// TIA Portal V16 export
// export: Created 2023-03-29T11:04:44.0584651Z, ExportSetting WithDefaults, DisplayName Totally Integrated Automation Portal, DisplayVersion V16 Update 6, DisplayName TIA Portal Version Control Interface, DisplayVersion V16 Update 2, DisplayName TIA Portal Openness, DisplayVersion V16 Update 6, DisplayName STEP 7 Professional, DisplayVersion V16 Update 6, DisplayName STEP 7 Safety, DisplayVersion V16, DisplayName WinCC Advanced, DisplayVersion V16 Update 6
FUNCTION_BLOCK "Kontrola przyrostu ciśnieniea"   // FB3, LAD
TITLE = Kalkulacja przyrostu ciśnienia w czasie
{ S7_Optimized_Access := 'TRUE' }
AUTHOR : RTecmer
FAMILY : PID
VERSION : 0.1
// Funkcja ustala czy następuje przyrost ciśnienia, spadek, równowaga. Pomiar dokonywany jest w ustalonym czasie. W zależności od wyliceń ustawiany jest znacznik, który w funkcji Switch_Motor_Extra dopuszcza lub blokuje uruchomienie dodatkowej pompy
// stored: AutoNumber true, IsIECCheckEnabled false, IsRetainMemResEnabled false, MemoryReserve 500, SetENOAutomatically false, UDAEnableTagReadback false
   VAR_INPUT
      "50Hz" : Bool;   // Znacznik 50Hz
      "Set_O2-PID" : Real;   // Zadana wartość ciśnienia [bar]
      Current_bar_1 : Real;   // aktualne ciśnienie
   END_VAR
   VAR_OUTPUT
      Increase_in_value : Bool;   // Wzwrost wartości bar w jednostce czasu
   END_VAR
   VAR_IN_OUT
      Edge1_Hz : Bool;   // Pamięć zbocza dla pierwszego odczytu
      Edge2_Hz : Bool;   // Pamięć zbocza dla drugiego odczytu
      Data_sek_1 : Int;   // Licznik sekund dla pierwszego odczytu
      Data_sek_2 : Int;   // Licznik sekund dla drugiego odczytu
      Pause_1 : Bool;   // Wstrzymanie dla pierwszego czasu
      Pause_2 : Bool;   // wstrzymanie dla drugiego czasu
   END_VAR
   VAR_TEMP   // added for the SCL form of the ladder/FBD networks
      _w1 : Bool;
      _w2 : Bool;
   END_VAR
BEGIN

REGION Network 1: Wstrzymanie dla pierwszego czasu
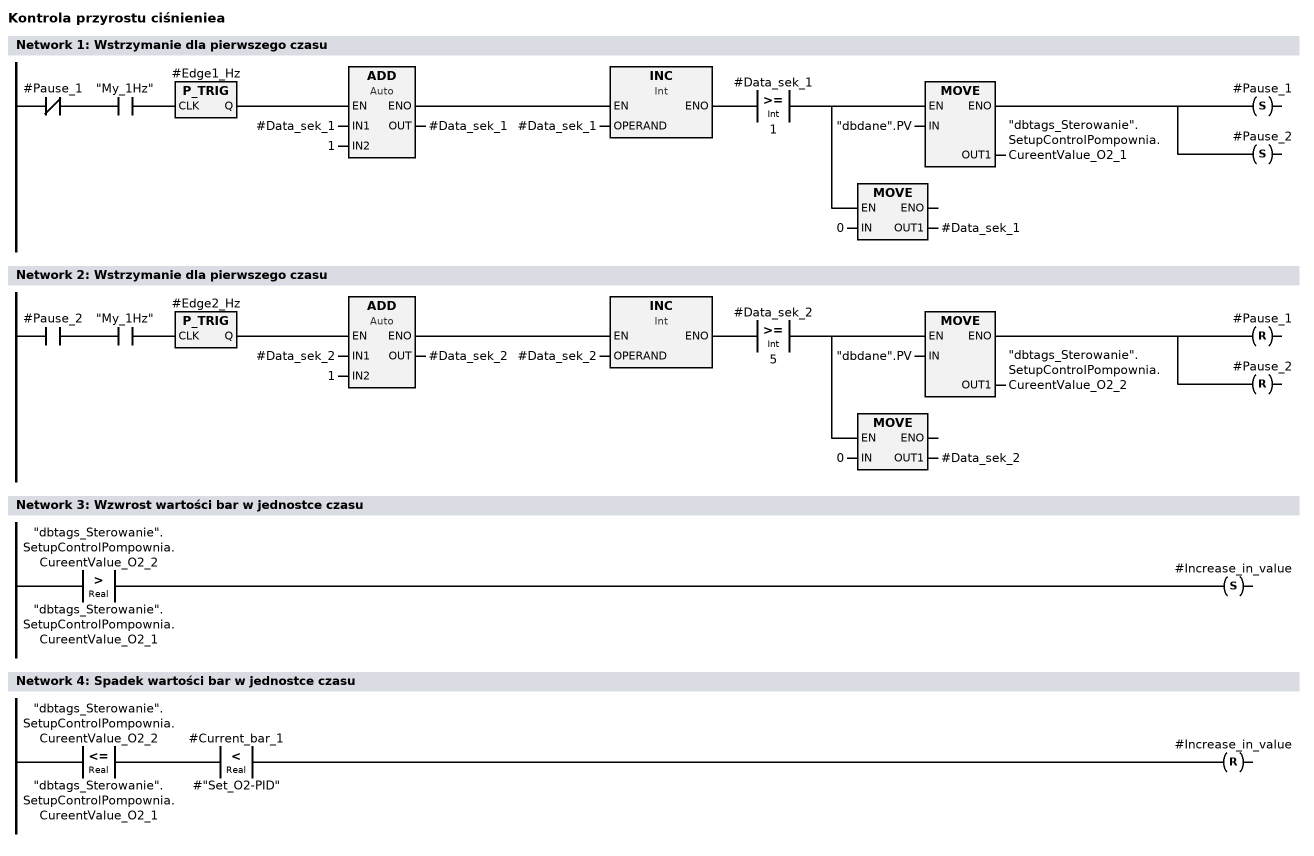
   RUNG wire#powerrail
      I_Contact( #Pause_1 )
      Contact( "My_1Hz" )
      P_Trig( #Edge1_Hz )
      { S7_GenerateENO := "TRUE" } Add(in1 := #Data_sek_1, in2 := 1, out => #Data_sek_1)
      { S7_Templates := "DestType := Int"; S7_GenerateENO := "TRUE" } Inc( #Data_sek_1 )
      { S7_Templates := "SrcType := Int" } GE_Contact(in1 := #Data_sek_1, in2 := 1)
      wire#w1
      { S7_GenerateENO := "TRUE" } Move(in := "dbdane".PV, out1 => "dbtags_Sterowanie".SetupControlPompownia.CureentValue_O2_1)
      wire#w2
      S_Coil( #Pause_1 )
   END_RUNG
   RUNG wire#w2
      S_Coil( #Pause_2 )
   END_RUNG
   RUNG wire#w1
      { S7_GenerateENO := "TRUE" } Move(in := 0, out1 => #Data_sek_1)
   END_RUNG
   // the same network as SCL:
   // ENO of a box is taken as its EN; it also drops when the box reports an error
   #_w1 := NOT #Pause_1 AND "My_1Hz";
   #_w2 := #_w1 AND NOT #Edge1_Hz;   // rising edge
   #Edge1_Hz := #_w1;
   IF #_w2 THEN
       #Data_sek_1 := #Data_sek_1 + 1;
       #Data_sek_1 := #Data_sek_1 + 1;
   END_IF;
   IF #_w2 AND (#Data_sek_1 >= 1) THEN
       "dbtags_Sterowanie".SetupControlPompownia.CureentValue_O2_1 := "dbdane".PV;
       #Pause_1 := TRUE;
       #Pause_2 := TRUE;
       #Data_sek_1 := 0;
   END_IF;
END_REGION

REGION Network 2: Wstrzymanie dla pierwszego czasu
   RUNG wire#powerrail
      Contact( #Pause_2 )
      Contact( "My_1Hz" )
      P_Trig( #Edge2_Hz )
      { S7_GenerateENO := "TRUE" } Add(in1 := #Data_sek_2, in2 := 1, out => #Data_sek_2)
      { S7_Templates := "DestType := Int"; S7_GenerateENO := "TRUE" } Inc( #Data_sek_2 )
      { S7_Templates := "SrcType := Int" } GE_Contact(in1 := #Data_sek_2, in2 := 5)
      wire#w1
      { S7_GenerateENO := "TRUE" } Move(in := "dbdane".PV, out1 => "dbtags_Sterowanie".SetupControlPompownia.CureentValue_O2_2)
      wire#w2
      R_Coil( #Pause_1 )
   END_RUNG
   RUNG wire#w2
      R_Coil( #Pause_2 )
   END_RUNG
   RUNG wire#w1
      { S7_GenerateENO := "TRUE" } Move(in := 0, out1 => #Data_sek_2)
   END_RUNG
   // the same network as SCL:
   // ENO of a box is taken as its EN; it also drops when the box reports an error
   #_w1 := #Pause_2 AND "My_1Hz";
   #_w2 := #_w1 AND NOT #Edge2_Hz;   // rising edge
   #Edge2_Hz := #_w1;
   IF #_w2 THEN
       #Data_sek_2 := #Data_sek_2 + 1;
       #Data_sek_2 := #Data_sek_2 + 1;
   END_IF;
   IF #_w2 AND (#Data_sek_2 >= 5) THEN
       "dbtags_Sterowanie".SetupControlPompownia.CureentValue_O2_2 := "dbdane".PV;
       #Pause_1 := FALSE;
       #Pause_2 := FALSE;
       #Data_sek_2 := 0;
   END_IF;
END_REGION

REGION Network 3: Wzwrost wartości bar w jednostce czasu
   RUNG wire#powerrail
      { S7_Templates := "SrcType := Real" } GT_Contact(in1 := "dbtags_Sterowanie".SetupControlPompownia.CureentValue_O2_2, in2 := "dbtags_Sterowanie".SetupControlPompownia.CureentValue_O2_1)
      S_Coil( #Increase_in_value )
   END_RUNG
   // the same network as SCL:
   IF "dbtags_Sterowanie".SetupControlPompownia.CureentValue_O2_2 > "dbtags_Sterowanie".SetupControlPompownia.CureentValue_O2_1 THEN
       #Increase_in_value := TRUE;
   END_IF;
END_REGION

REGION Network 4: Spadek wartości bar w jednostce czasu
   RUNG wire#powerrail
      { S7_Templates := "SrcType := Real" } LE_Contact(in1 := "dbtags_Sterowanie".SetupControlPompownia.CureentValue_O2_2, in2 := "dbtags_Sterowanie".SetupControlPompownia.CureentValue_O2_1)
      { S7_Templates := "SrcType := Real" } LT_Contact(in1 := #Current_bar_1, in2 := #"Set_O2-PID")
      R_Coil( #Increase_in_value )
   END_RUNG
   // the same network as SCL:
   IF ("dbtags_Sterowanie".SetupControlPompownia.CureentValue_O2_2 <= "dbtags_Sterowanie".SetupControlPompownia.CureentValue_O2_1) AND (#Current_bar_1 < #"Set_O2-PID") THEN
       #Increase_in_value := FALSE;
   END_IF;
END_REGION
END_FUNCTION_BLOCK
